// SIMATIC STEP 7 (V5.x) project nef
// CPU: PLC 314C-2 DP
// station: P_ADR_BUS
// station: Hardware
// station: SIMATIC 300(1)
// program: Programma S7(1)

SYMBOL_TABLE
"READ_CLK"	SFC 1	SFC 1	// Read System Clock
"BLKMOV"	SFC 20	SFC 20	// Copy Variables
"FILL"	SFC 21	SFC 21	// Initialize a Memory Area
"CREAT_DB"	SFC 22	SFC 22	// Create Data Block
"DIS_AIRT"	SFC 41	SFC 41	// Delay the Higher Priority Interrupts and Asynchronous Errors
"EN_AIRT"	SFC 42	SFC 42	// Enable Higher Priority Interrupts and Asynchronous Errors
"STP"	SFC 46	SFC 46	// Change the CPU to STOP
"WAIT"	SFC 47	SFC 47	// Delay Execution of the User Program
"RDSYSST"	SFC 51	SFC 51	// Read a System Status List or Partial List
"WR_USMSG"	SFC 52	SFC 52	// Write a User-Defined Diagnostic Event to the Diagnostic Buffer
"TIME_TCK"	SFC 64	SFC 64	// Read the System Time
END_SYMBOL_TABLE

// FB 1: know-how protected block, not included

// FB 2: know-how protected block, not included

// FB 3: know-how protected block, not included

// FB 4: know-how protected block, not included

// FB 5: know-how protected block, not included

// FB 6: know-how protected block, not included

// FB 7: know-how protected block, not included

// FB 9: know-how protected block, not included

// FB 10: know-how protected block, not included

// FB 11: know-how protected block, not included

// FB 15: know-how protected block, not included

// FB 16: know-how protected block, not included

// FB 17: know-how protected block, not included

// FB 18: know-how protected block, not included

// FB 19: know-how protected block, not included

FUNCTION_BLOCK FB 20
VERSION : 2.2
BEGIN
// (block stored without names or comments; labels and parameter names are numbered)
NETWORK
TITLE =
      L     DW#16#87000000;
      LAR1;
      L     80;
      L     W#16#A000;
      +I;
      T     LW 0;
      A      [AR1,P#8.0];
      =     L 0.0;
      L     W [AR1,P#0.0];
      T     LW 2;
      L     W [AR1,P#6.0];
      SLD   16;
      L     B [AR1,P#4.0];
      OD;
      T     LD 4;
      CALL  "WR_USMSG" (
           SEND                     := TRUE,
           EVENTN                   := LW 0,
           INFO1                    := P#L 2.0 INT 1,
           INFO2                    := P#L 4.0 DINT 1,
           RET_VAL                  := LW 8);
END_FUNCTION_BLOCK

FUNCTION_BLOCK FB 100
VERSION : 0.0
BEGIN
// body was compiled from an SCL source; compiled code not shown
END_FUNCTION_BLOCK

FUNCTION_BLOCK FB 101
VERSION : 0.0
BEGIN
// body was compiled from an SCL source; compiled code not shown
END_FUNCTION_BLOCK

// FB 102: know-how protected block, not included

FUNCTION_BLOCK FB 103
VERSION : 0.0
BEGIN
// body was compiled from an SCL source; compiled code not shown
END_FUNCTION_BLOCK

// FB 104: know-how protected block, not included

FUNCTION_BLOCK FB 106
VERSION : 0.0
BEGIN
// body was compiled from an SCL source; compiled code not shown
END_FUNCTION_BLOCK

FUNCTION_BLOCK FB 107
VERSION : 0.0
BEGIN
// body was compiled from an SCL source; compiled code not shown
END_FUNCTION_BLOCK

FUNCTION_BLOCK FB 108
VERSION : 0.0
BEGIN
// body was compiled from an SCL source; compiled code not shown
END_FUNCTION_BLOCK

FUNCTION_BLOCK FB 109
VERSION : 0.0
BEGIN
// body was compiled from an SCL source; compiled code not shown
END_FUNCTION_BLOCK

FUNCTION_BLOCK FB 110
VERSION : 0.0
BEGIN
// body was compiled from an SCL source; compiled code not shown
END_FUNCTION_BLOCK

FUNCTION_BLOCK FB 111
VERSION : 0.0
BEGIN
// body was compiled from an SCL source; compiled code not shown
END_FUNCTION_BLOCK

FUNCTION_BLOCK FB 114
VERSION : 0.0
BEGIN
// body was compiled from an SCL source; compiled code not shown
END_FUNCTION_BLOCK

FUNCTION_BLOCK FB 115
VERSION : 0.0
BEGIN
// body was compiled from an SCL source; compiled code not shown
END_FUNCTION_BLOCK

// FB 116: know-how protected block, not included

FUNCTION_BLOCK FB 117
VERSION : 0.0
BEGIN
// body was compiled from an SCL source; compiled code not shown
END_FUNCTION_BLOCK

FUNCTION_BLOCK FB 118
VERSION : 0.0
BEGIN
// body was compiled from an SCL source; compiled code not shown
END_FUNCTION_BLOCK

FUNCTION_BLOCK FB 119
VERSION : 0.0
BEGIN
// body was compiled from an SCL source; compiled code not shown
END_FUNCTION_BLOCK

FUNCTION_BLOCK FB 120
VERSION : 0.0
BEGIN
// body was compiled from an SCL source; compiled code not shown
END_FUNCTION_BLOCK

// FB 122: know-how protected block, not included

FUNCTION_BLOCK FB 123
VERSION : 0.0
BEGIN
// body was compiled from an SCL source; compiled code not shown
END_FUNCTION_BLOCK

FUNCTION_BLOCK FB 124
VERSION : 0.0
BEGIN
// body was compiled from an SCL source; compiled code not shown
END_FUNCTION_BLOCK

FUNCTION_BLOCK FB 125
VERSION : 0.0
BEGIN
// body was compiled from an SCL source; compiled code not shown
END_FUNCTION_BLOCK

FUNCTION_BLOCK FB 126
VERSION : 0.0
BEGIN
// body was compiled from an SCL source; compiled code not shown
END_FUNCTION_BLOCK

FUNCTION_BLOCK FB 127
VERSION : 0.0
BEGIN
// body was compiled from an SCL source; compiled code not shown
END_FUNCTION_BLOCK

FUNCTION_BLOCK FB 131
VERSION : 0.0
BEGIN
// body was compiled from an SCL source; compiled code not shown
END_FUNCTION_BLOCK

FUNCTION_BLOCK FB 132
VERSION : 0.0
BEGIN
// body was compiled from an SCL source; compiled code not shown
END_FUNCTION_BLOCK

FUNCTION_BLOCK FB 133
VERSION : 0.0
BEGIN
// body was compiled from an SCL source; compiled code not shown
END_FUNCTION_BLOCK

FUNCTION_BLOCK FB 135
VERSION : 0.0
BEGIN
// body was compiled from an SCL source; compiled code not shown
END_FUNCTION_BLOCK

FUNCTION_BLOCK FB 138
VERSION : 0.0
BEGIN
// body was compiled from an SCL source; compiled code not shown
END_FUNCTION_BLOCK

FUNCTION_BLOCK FB 144
VERSION : 0.0
BEGIN
// body was compiled from an SCL source; compiled code not shown
END_FUNCTION_BLOCK

FUNCTION_BLOCK FB 148
VERSION : 0.0
BEGIN
// body was compiled from an SCL source; compiled code not shown
END_FUNCTION_BLOCK

FUNCTION_BLOCK FB 189
AUTHOR : mogs
NAME : s_remind
VERSION : 1.3
BEGIN
// (block stored without names or comments; labels and parameter names are numbered)
NETWORK
TITLE =
      A     DIX 1.0;
      =     L 12.0;
      A     L 12.0;
      A     DIX 172.1;
      R     DIX 172.1;
      R     DIX 173.0;
      A     L 12.0;
      A     DIX 172.0;
      R     DIX 172.0;
      R     DIX 172.7;
      A     L 12.0;
      BLD   102;
      R     DIX 172.2;
NETWORK
TITLE =
      A     DIX 1.1;
      =     L 12.0;
      A     L 12.0;
      A     DIX 172.1;
      R     DIX 172.1;
      S     DIX 173.0;
      A     L 12.0;
      A     DIX 172.0;
      S     DIX 172.7;
      R     DIX 172.0;
      A     L 12.0;
      BLD   102;
      R     DIX 172.3;
NETWORK
TITLE =
      A     DIX 172.0;
      A(;
      L     DIW 2;
      L     0;
      >I;
      );
      =     DIX 18.0;
NETWORK
TITLE =
      A     DIX 172.1;
      A(;
      L     DIW 2;
      L     0;
      >I;
      );
      =     DIX 18.1;
NETWORK
TITLE =
      A     DIX 0.0;
      FP    DIX 172.6;
      =     L 12.0;
      A     L 12.0;
      A     DIX 172.7;
      S     DIX 172.0;
      A     L 12.0;
      A     DIX 173.0;
      S     DIX 172.1;
NETWORK
TITLE =
      BLD   7;
      L     0;
      T     LW 13;
      L     P#V 0.0;
      T     LD 15;
      UC    "READ_CLK";
      {     P#L 8.0, P#L 13.0 };
      BLD   8;
      CLR;
      =     L 10.2;
      =     DIX 173.2;
      =     L 10.1;
      L     LB 5;
      L     DIB 59;
      ==I;
      JC    M001;
      TAK;
      T     DIB 59;
      =     L 10.2;
M001: L     LB 4;
      L     DIB 55;
      ==I;
      JC    M002;
      TAK;
      T     DIB 55;
      =     DIX 173.2;
M002: L     LB 3;
      L     DIB 54;
      ==I;
      JC    M003;
      T     DIB 54;
      =     L 10.1;
M003: L     LB 4;
      BTI;
      T     DIB 65;
      L     LB 3;
      BTI;
      T     DIB 64;
      L     LB 2;
      BTI;
      T     DIB 63;
      L     LB 1;
      BTI;
      T     DIB 62;
      L     LB 0;
      BTI;
      T     DIB 61;
      AN    L 10.2;
      AN    DIX 173.2;
      AN    L 10.1;
      BEC;
NETWORK
TITLE =
// (network holds code this reader does not know; not shown)
NETWORK
TITLE =
// (network holds code this reader does not know; not shown)
NETWORK
TITLE =
// (network holds code this reader does not know; not shown)
NETWORK
TITLE =
M009: NOP   0;
NETWORK
TITLE =
      A     DIX 173.1;
      =     L 12.0;
      A     L 12.0;
      A     DIX 0.3;
      JNB   M010;
      L     0;
      T     DIW 72;
      SET;
      SAVE;
      CLR;
M010: A     BR;
      S     DIX 172.5;
      R     DIX 0.3;
      A     L 12.0;
      A     DIX 172.5;
      A(;
      L     DIW 72;
      L     DIW 4;
      >=I;
      );
      R     DIX 172.5;
NETWORK
TITLE =
      A     DIX 172.5;
      A     DIX 0.0;
      A     DIX 173.2;
      JNB   M011;
      L     DIW 72;
      L     1;
      +I;
      T     DIW 72;
M011: NOP   0;
NETWORK
TITLE =
      BEU;
END_FUNCTION_BLOCK

FUNCTION_BLOCK FB 201
AUTHOR : Duesed
NAME : M_Dek
VERSION : 0.1
BEGIN
// (block stored without names or comments; labels and parameter names are numbered)
NETWORK
TITLE =
      A     DIX [AR2,P#6.0];
      JC    M001;
      JU    M003;
M001: T     LD 27;
      TAK;
      T     LD 31;
      L     DIW [AR2,P#4.0];
      T     LW 35;
      L     LD 31;
      L     LD 27;
      OPN   DB [LW 35];
      L     P#0.0;
      LAR1;
      L     95;
M002: T     LW 4;
      L     0;
      T     DBD [AR1,P#0.0];
      +AR1  P#4.0;
      L     LW 4;
      LOOP  M002;
      CLR;
      =     DIX [AR2,P#8.0];
      =     DIX [AR2,P#8.1];
      =     DIX [AR2,P#8.2];
      L     0;
      T     DID [AR2,P#30.0];
      T     DID [AR2,P#34.0];
      T     DID [AR2,P#38.0];
      T     DID [AR2,P#42.0];
      T     DID [AR2,P#46.0];
      L     -1;
      T     DIW [AR2,P#20.0];
      T     DIW [AR2,P#22.0];
      T     DIW [AR2,P#24.0];
      T     DIW [AR2,P#26.0];
      T     DIW [AR2,P#28.0];
M003: A     DIX [AR2,P#6.1];
      JCN   M032;
      R     DIX [AR2,P#8.4];
      L     -1;
      T     DIW [AR2,P#10.0];
      T     DIW [AR2,P#12.0];
      T     DIW [AR2,P#14.0];
      T     DIW [AR2,P#16.0];
      T     DIW [AR2,P#18.0];
      T     LD 27;
      TAK;
      T     LD 31;
      L     DIW [AR2,P#4.0];
      T     LW 35;
      L     LD 31;
      L     LD 27;
      OPN   DB [LW 35];
      L     0;
      T     LW 24;
M004: L     LW 24;
      JL    M005;
      JU    M006;
      JU    M007;
      JU    M008;
      JU    M009;
      JU    M010;
M005: CLR;
      =     L 26.1;
      JU    M013;
M006: CLR;
      =     L 26.1;
      L     DIW [AR2,P#20.0];
      L     DIW [AR2,P#22.0];
      ==I;
      S     L 26.1;
      L     DIW [AR2,P#20.0];
      L     DIW [AR2,P#24.0];
      ==I;
      S     L 26.1;
      L     DIW [AR2,P#20.0];
      L     DIW [AR2,P#26.0];
      ==I;
      S     L 26.1;
      L     DIW [AR2,P#20.0];
      L     DIW [AR2,P#28.0];
      ==I;
      S     L 26.1;
      L     DIW [AR2,P#20.0];
      T     LD 20;
      L     DID [AR2,P#30.0];
      T     LD 14;
      JU    M011;
M007: CLR;
      =     L 26.1;
      L     DIW [AR2,P#22.0];
      L     DIW [AR2,P#24.0];
      ==I;
      S     L 26.1;
      L     DIW [AR2,P#22.0];
      L     DIW [AR2,P#26.0];
      ==I;
      S     L 26.1;
      L     DIW [AR2,P#22.0];
      L     DIW [AR2,P#28.0];
      ==I;
      S     L 26.1;
      L     DIW [AR2,P#22.0];
      T     LD 20;
      L     DID [AR2,P#34.0];
      T     LD 14;
      JU    M011;
M008: CLR;
      =     L 26.1;
      L     DIW [AR2,P#24.0];
      L     DIW [AR2,P#26.0];
      ==I;
      S     L 26.1;
      L     DIW [AR2,P#24.0];
      L     DIW [AR2,P#28.0];
      ==I;
      S     L 26.1;
      L     DIW [AR2,P#24.0];
      T     LD 20;
      L     DID [AR2,P#38.0];
      T     LD 14;
      JU    M011;
M009: CLR;
      =     L 26.1;
      L     DIW [AR2,P#26.0];
      L     DIW [AR2,P#28.0];
      ==I;
      S     L 26.1;
      L     DIW [AR2,P#26.0];
      T     LD 20;
      L     DID [AR2,P#42.0];
      T     LD 14;
      JU    M011;
M010: CLR;
      =     L 26.1;
      L     DIW [AR2,P#28.0];
      T     LD 20;
      L     DID [AR2,P#46.0];
      T     LD 14;
      JU    M011;
NETWORK
TITLE =
M011: L     LD 20;
      L     -1;
      ==I;
      JC    M012;
      A     L 26.1;
      S     DIX [AR2,P#8.3];
      JC    M012;
      L     LD 20;
      L     999;
      >I;
      JC    M012;
M012: L     LW 24;
      INC   1;
      T     LW 24;
      JU    M004;
M013: NOP   0;
NETWORK
TITLE =
      L     0;
      T     LW 24;
M014: L     LW 24;
      JL    M015;
      JU    M016;
      JU    M017;
      JU    M018;
      JU    M019;
      JU    M020;
M015: BEU;
M016: T     LD 27;
      TAK;
      T     LD 31;
      L     DIW [AR2,P#0.0];
      T     LW 35;
      L     LD 31;
      L     LD 27;
      OPN   DB [LW 35];
      A     DBX 66.0;
      =     L 26.0;
      AN    DBX 58.0;
      JC    M031;
      L     DBW 68;
      T     LW 18;
      L     DBD 70;
      T     LD 20;
      JU    M021;
M017: T     LD 27;
      TAK;
      T     LD 31;
      L     DIW [AR2,P#0.0];
      T     LW 35;
      L     LD 31;
      L     LD 27;
      OPN   DB [LW 35];
      A     DBX 66.1;
      =     L 26.0;
      AN    DBX 58.1;
      JC    M031;
      L     DBW 74;
      T     LW 18;
      L     DBD 76;
      T     LD 20;
      JU    M021;
M018: T     LD 27;
      TAK;
      T     LD 31;
      L     DIW [AR2,P#0.0];
      T     LW 35;
      L     LD 31;
      L     LD 27;
      OPN   DB [LW 35];
      A     DBX 66.2;
      =     L 26.0;
      AN    DBX 58.2;
      JC    M031;
      L     DBW 80;
      T     LW 18;
      L     DBD 82;
      T     LD 20;
      JU    M021;
M019: T     LD 27;
      TAK;
      T     LD 31;
      L     DIW [AR2,P#0.0];
      T     LW 35;
      L     LD 31;
      L     LD 27;
      OPN   DB [LW 35];
      A     DBX 66.3;
      =     L 26.0;
      AN    DBX 58.3;
      JC    M031;
      L     DBW 86;
      T     LW 18;
      L     DBD 88;
      T     LD 20;
      JU    M021;
M020: T     LD 27;
      TAK;
      T     LD 31;
      L     DIW [AR2,P#0.0];
      T     LW 35;
      L     LD 31;
      L     LD 27;
      OPN   DB [LW 35];
      A     DBX 66.4;
      =     L 26.0;
      AN    DBX 58.4;
      JC    M031;
      L     DBW 92;
      T     LW 18;
      L     DBD 94;
      T     LD 20;
      JU    M021;
NETWORK
TITLE =
M021: L     LW 18;
      L     0;
      ==I;
      JC    M024;
      L     LW 18;
      L     DIW [AR2,P#2.0];
      >I;
      JC    M022;
      L     LD 20;
      L     3;
      ==I;
      JC    M023;
      L     LD 20;
      L     4;
      ==I;
      JC    M023;
      L     LD 20;
      L     5;
      ==I;
      JC    M023;
      L     LD 20;
      L     40;
      ==I;
      JC    M023;
      L     LD 20;
      L     41;
      ==I;
      JC    M023;
      L     LD 20;
      L     42;
      ==I;
      JC    M023;
      L     LD 20;
      L     70;
      ==I;
      JC    M031;
M022: S     DIX [AR2,P#8.2];
      JU    M031;
M023: L     LW 18;
      L     100;
      *I;
      L     LD 20;
      +I;
      T     LD 20;
M024: L     LD 20;
      L     999;
      >D;
      S     DIX [AR2,P#8.1];
      JC    M031;
      L     LD 20;
      L     8;
      /I;
      T     LD 6;
      L     LD 6;
      SLD   16;
      SRD   16;
      T     LW 10;
      L     LD 6;
      SRD   16;
      T     LW 12;
      L     LW 10;
      SLW   3;
      L     LW 12;
      OW;
      L     DW#16#4000000;
      OW;
      LAR1;
      T     LD 14;
      T     LD 27;
      TAK;
      T     LD 31;
      L     DIW [AR2,P#4.0];
      T     LW 35;
      L     LD 31;
      L     LD 27;
      OPN   DB [LW 35];
      SET;
      =     DBX [AR1,P#0.0];
      S     DIX [AR2,P#8.4];
      A     L 26.0;
      =     DBX [AR1,P#252.0];
      L     LW 24;
      JL    M025;
      JU    M026;
      JU    M027;
      JU    M028;
      JU    M029;
      JU    M030;
M025: JU    M031;
M026: L     LD 14;
      T     DID [AR2,P#30.0];
      L     LD 20;
      T     DIW [AR2,P#20.0];
      T     DIW [AR2,P#10.0];
      JU    M031;
M027: L     LD 14;
      T     DID [AR2,P#34.0];
      L     LD 20;
      T     DIW [AR2,P#22.0];
      T     DIW [AR2,P#12.0];
      JU    M031;
M028: L     LD 14;
      T     DID [AR2,P#38.0];
      L     LD 20;
      T     DIW [AR2,P#24.0];
      T     DIW [AR2,P#14.0];
      JU    M031;
M029: L     LD 14;
      T     DID [AR2,P#42.0];
      L     LD 20;
      T     DIW [AR2,P#26.0];
      T     DIW [AR2,P#16.0];
      JU    M031;
M030: L     LD 14;
      T     DID [AR2,P#46.0];
      L     LD 20;
      T     DIW [AR2,P#28.0];
      T     DIW [AR2,P#18.0];
      JU    M031;
M031: L     LW 24;
      INC   1;
      T     LW 24;
      JU    M014;
M032: NOP   0;
NETWORK
TITLE =
      AN    DIX [AR2,P#6.1];
      JCN   M038;
      L     DIW [AR2,P#20.0];
      L     -1;
      ==I;
      JC    M033;
      TAK;
      L     999;
      >I;
      JC    M033;
      T     LD 27;
      TAK;
      T     LD 31;
      L     DIW [AR2,P#4.0];
      T     LW 35;
      L     LD 31;
      L     LD 27;
      OPN   DB [LW 35];
      L     DID [AR2,P#30.0];
      LAR1;
      AN    DBX [AR1,P#126.0];
      S     DIX [AR2,P#8.0];
      CLR;
      =     DBX [AR1,P#0.0];
      =     DBX [AR1,P#126.0];
      =     DBX [AR1,P#252.0];
M033: NOP   0;
      L     0;
      T     DID [AR2,P#30.0];
      L     -1;
      T     DIW [AR2,P#20.0];
      L     DIW [AR2,P#22.0];
      L     -1;
      ==I;
      JC    M034;
      TAK;
      L     999;
      >I;
      JC    M034;
      T     LD 27;
      TAK;
      T     LD 31;
      L     DIW [AR2,P#4.0];
      T     LW 35;
      L     LD 31;
      L     LD 27;
      OPN   DB [LW 35];
      L     DID [AR2,P#34.0];
      LAR1;
      AN    DBX [AR1,P#126.0];
      S     DIX [AR2,P#8.0];
      CLR;
      =     DBX [AR1,P#0.0];
      =     DBX [AR1,P#126.0];
      =     DBX [AR1,P#252.0];
M034: NOP   0;
      L     0;
      T     DID [AR2,P#34.0];
      L     -1;
      T     DIW [AR2,P#22.0];
      L     DIW [AR2,P#24.0];
      L     -1;
      ==I;
      JC    M035;
      TAK;
      L     999;
      >I;
      JC    M035;
      T     LD 27;
      TAK;
      T     LD 31;
      L     DIW [AR2,P#4.0];
      T     LW 35;
      L     LD 31;
      L     LD 27;
      OPN   DB [LW 35];
      L     DID [AR2,P#38.0];
      LAR1;
      AN    DBX [AR1,P#126.0];
      S     DIX [AR2,P#8.0];
      CLR;
      =     DBX [AR1,P#0.0];
      =     DBX [AR1,P#126.0];
      =     DBX [AR1,P#252.0];
M035: NOP   0;
      L     0;
      T     DID [AR2,P#38.0];
      L     -1;
      T     DIW [AR2,P#24.0];
      L     DIW [AR2,P#26.0];
      L     -1;
      ==I;
      JC    M036;
      TAK;
      L     999;
      >I;
      JC    M036;
      T     LD 27;
      TAK;
      T     LD 31;
      L     DIW [AR2,P#4.0];
      T     LW 35;
      L     LD 31;
      L     LD 27;
      OPN   DB [LW 35];
      L     DID [AR2,P#42.0];
      LAR1;
      AN    DBX [AR1,P#126.0];
      S     DIX [AR2,P#8.0];
      CLR;
      =     DBX [AR1,P#0.0];
      =     DBX [AR1,P#126.0];
      =     DBX [AR1,P#252.0];
M036: NOP   0;
      L     0;
      T     DID [AR2,P#42.0];
      L     -1;
      T     DIW [AR2,P#26.0];
      L     DIW [AR2,P#28.0];
      L     -1;
      ==I;
      JC    M037;
      TAK;
      L     999;
      >I;
      JC    M037;
      T     LD 27;
      TAK;
      T     LD 31;
      L     DIW [AR2,P#4.0];
      T     LW 35;
      L     LD 31;
      L     LD 27;
      OPN   DB [LW 35];
      L     DID [AR2,P#46.0];
      LAR1;
      AN    DBX [AR1,P#126.0];
      S     DIX [AR2,P#8.0];
      CLR;
      =     DBX [AR1,P#0.0];
      =     DBX [AR1,P#126.0];
      =     DBX [AR1,P#252.0];
M037: NOP   0;
      L     0;
      T     DID [AR2,P#46.0];
      L     -1;
      T     DIW [AR2,P#28.0];
M038: NOP   0;
END_FUNCTION_BLOCK

FUNCTION_BLOCK FB 203
VERSION : 0.0
BEGIN
// body was compiled from an SCL source; compiled code not shown
END_FUNCTION_BLOCK

FUNCTION_BLOCK FB 204
VERSION : 0.0
BEGIN
// body was compiled from an SCL source; compiled code not shown
END_FUNCTION_BLOCK

FUNCTION_BLOCK FB 205
VERSION : 0.0
BEGIN
// body was compiled from an SCL source; compiled code not shown
END_FUNCTION_BLOCK

FUNCTION_BLOCK FB 206
VERSION : 0.0
BEGIN
// body was compiled from an SCL source; compiled code not shown
END_FUNCTION_BLOCK

FUNCTION_BLOCK FB 208
VERSION : 0.0
BEGIN
// body was compiled from an SCL source; compiled code not shown
END_FUNCTION_BLOCK

FUNCTION_BLOCK FB 209
VERSION : 0.0
BEGIN
// body was compiled from an SCL source; compiled code not shown
END_FUNCTION_BLOCK

FUNCTION_BLOCK FB 214
AUTHOR : BI_HSc
VERSION : 0.1
BEGIN
// (block stored without names or comments; labels and parameter names are numbered)
NETWORK
TITLE =
      A     M 0.5;
      JCN   M001;
      OPN   DB 2;
      L     DBLG;
      L     180;
      -I;
      L     8;
      /I;
      OPN   DB 214;
      T     DIW [AR2,P#160.0];
M001: NOP   0;
NETWORK
TITLE =
      OPN   DB 2;
      L     P#180.0;
      LAR1;
      L     P#0.0;
      OPN   DB 214;
      L     P#0.0;
      LAR2;
      SET;
      R     M 2.3;
      R     M 2.4;
      R     M 2.6;
      R     M 2.7;
      R     M 3.0;
      L     DIW [AR2,P#160.0];
M002: T     LW 0;
      OPN   DB 2;
      L     DBD [AR1,P#0.0];
      T     LD 2;
      L     0;
      <>D;
      S     M 2.3;
      TAK;
      OPN   DB 214;
      L     DBD [AR2,P#0.0];
      XOD;
      L     LD 2;
      AD;
      L     0;
      <>D;
      S     M 2.6;
      L     LD 2;
      T     DBD [AR2,P#0.0];
      +AR1  P#4.0;
      +AR2  P#4.0;
      OPN   DB 2;
      L     DBD [AR1,P#0.0];
      T     LD 2;
      L     0;
      <>D;
      S     M 2.4;
      TAK;
      OPN   DB 214;
      L     DBD [AR2,P#0.0];
      XOD;
      L     LD 2;
      AD;
      L     0;
      <>D;
      S     M 2.7;
      L     LD 2;
      T     DBD [AR2,P#0.0];
      +AR1  P#4.0;
      +AR2  P#4.0;
      L     LW 0;
      LOOP  M002;
      A     DB10.DBX 109.0;
      AN    M 2.5;
      S     M 3.0;
      A     DB10.DBX 109.0;
      =     M 2.5;
END_FUNCTION_BLOCK

FUNCTION_BLOCK FB 219
VERSION : 0.0
BEGIN
// body was compiled from an SCL source; compiled code not shown
END_FUNCTION_BLOCK

FUNCTION_BLOCK FB 220
VERSION : 0.0
BEGIN
// body was compiled from an SCL source; compiled code not shown
END_FUNCTION_BLOCK

FUNCTION_BLOCK FB 221
VERSION : 0.0
BEGIN
// body was compiled from an SCL source; compiled code not shown
END_FUNCTION_BLOCK

FUNCTION_BLOCK FB 240
VERSION : 0.0
BEGIN
// body was compiled from an SCL source; compiled code not shown
END_FUNCTION_BLOCK

FUNCTION_BLOCK FB 250
VERSION : 0.0
BEGIN
// body was compiled from an SCL source; compiled code not shown
END_FUNCTION_BLOCK

FUNCTION_BLOCK FB 252
VERSION : 0.0
BEGIN
// body was compiled from an SCL source; compiled code not shown
END_FUNCTION_BLOCK

FUNCTION_BLOCK FB 253
VERSION : 0.0
BEGIN
// body was compiled from an SCL source; compiled code not shown
END_FUNCTION_BLOCK

// FC 1: know-how protected block, not included

// FC 2: know-how protected block, not included

// FC 3: know-how protected block, not included

// FC 4: know-how protected block, not included

// FC 6: know-how protected block, not included

// FC 7: know-how protected block, not included

// FC 8: know-how protected block, not included

// FC 9: know-how protected block, not included

// FC 10: know-how protected block, not included

// FC 11: know-how protected block, not included

FUNCTION FC 12 : VOID
AUTHOR : NUMERIK
FAMILY : _800D
NAME : Basics
VERSION : 4.0
BEGIN
// (block stored without names or comments; labels and parameter names are numbered)
END_FUNCTION

// FC 13: know-how protected block, not included

// FC 14: know-how protected block, not included

// FC 15: know-how protected block, not included

// FC 16: know-how protected block, not included

// FC 17: know-how protected block, not included

// FC 18: know-how protected block, not included

FUNCTION FC 19 : VOID
AUTHOR : NUMERIK
FAMILY : _800D
NAME : MCP_IFM
VERSION : 6.1
BEGIN
// (block stored without names or comments; labels and parameter names are numbered)
NETWORK
TITLE =
// (network holds code this reader does not know; not shown)
END_FUNCTION

// FC 20: know-how protected block, not included

// FC 21: know-how protected block, not included

// FC 22: know-how protected block, not included

FUNCTION FC 24 : VOID
AUTHOR : NUMERIK
FAMILY : _800D
NAME : MCP_IFM2
VERSION : 6.1
BEGIN
// (block stored without names or comments; labels and parameter names are numbered)
NETWORK
TITLE =
// (network holds code this reader does not know; not shown)
END_FUNCTION

FUNCTION FC 25 : VOID
AUTHOR : NUMERIK
FAMILY : _800D
NAME : MCP_IFT
VERSION : 6.1
BEGIN
// (block stored without names or comments; labels and parameter names are numbered)
NETWORK
TITLE =
// (network holds code this reader does not know; not shown)
END_FUNCTION

FUNCTION FC 26 : VOID
AUTHOR : NUMERIK
FAMILY : _800D
NAME : HPU_MCP
VERSION : 6.2
BEGIN
// (block stored without names or comments; labels and parameter names are numbered)
NETWORK
TITLE =
// (network holds code this reader does not know; not shown)
END_FUNCTION

FUNCTION FC 30 : VOID
VERSION : 0.0
BEGIN
// body was compiled from another editor; compiled code not shown
END_FUNCTION

FUNCTION FC 31 : VOID
VERSION : 0.0
BEGIN
// body was compiled from another editor; compiled code not shown
END_FUNCTION

FUNCTION FC 32 : VOID
VERSION : 0.0
BEGIN
// body was compiled from another editor; compiled code not shown
END_FUNCTION

FUNCTION FC 33 : VOID
VERSION : 0.0
BEGIN
// body was compiled from another editor; compiled code not shown
END_FUNCTION

// FC 34: know-how protected block, not included

// FC 35: know-how protected block, not included

FUNCTION FC 119 : VOID
VERSION : 0.0
BEGIN
// body was compiled from an SCL source; compiled code not shown
END_FUNCTION

FUNCTION FC 123 : VOID
NAME : TEST2
VERSION : 0.0
BEGIN
// (block stored without names or comments; labels and parameter names are numbered)
NETWORK
TITLE =
      CLR;
      =     #PARAM7;
      L     0;
      T     #PARAM8;
      AN    #PARAM1;
      BEC;
      SET;
      S     L 0.0;
      L     -1;
      T     #PARAM6;
NETWORK
TITLE =
      L     #PARAM3;
      T     LW 2;
      OPN   DB [LW 2];
      L     DBLG;
      L     2;
      -D;
      T     LW 4;
      L     #PARAM4;
      L     LW 4;
      >D;
      L     2;
      JC    M002;
      A     #PARAM2;
      JC    M001;
NETWORK
TITLE =
      L     #PARAM4;
      SLW   3;
      LAR1;
      L     DBW [AR1,P#0.0];
      T     LW 6;
      T     #PARAM6;
      CALL  FC 21 (
           $1                       := P#L 0.0,
           $2                       := B#16#4,
           $3                       := P#L 6.0 WORD 1,
           $4                       := 1020,
           $5                       := -1,
           $6                       := #PARAM7,
           $7                       := #PARAM8);
      L     #PARAM8;
      A     #PARAM7;
      JC    M002;
      JU    M003;
NETWORK
TITLE =
M001: L     #PARAM4;
      SLW   3;
      LAR1;
      L     #PARAM5;
      T     DBW [AR1,P#0.0];
      JU    M003;
NETWORK
TITLE =
M002: SET;
      =     #PARAM7;
      T     #PARAM8;
M003: NOP   0;
END_FUNCTION

FUNCTION FC 200 : VOID
VERSION : 0.0
BEGIN
// body was compiled from an SCL source; compiled code not shown
END_FUNCTION

FUNCTION FC 201 : VOID
VERSION : 0.0
BEGIN
// body was compiled from an SCL source; compiled code not shown
END_FUNCTION

// FC 202: know-how protected block, not included

// FC 225: know-how protected block, not included

// FC 226: know-how protected block, not included

FUNCTION FC 241 : VOID
AUTHOR : RuestGeh
FAMILY : SPL
VERSION : 3.0
BEGIN
// (block stored without names or comments; labels and parameter names are numbered)
NETWORK
TITLE =
      L     P##PARAM4;
      LAR1;
      L     P##PARAM13;
      LAR2;
      L     DB5.DBW 24;
      L     #PARAM3;
      <I;
      JC    M054;
      L     0;
      >I;
      JCN   M054;
      TAK;
      L     8;
      >I;
      JC    M054;
      A     #PARAM14;
      R     #PARAM14;
      A     #PARAM2;
      FP     [AR2,P#1.6];
      JC    M055;
      A     #PARAM1;
      FP     [AR2,P#1.7];
      S      [AR2,P#0.0];
      L     P##PARAM4;
      LAR1;
      L     #PARAM3;
      A      [AR2,P#0.0];
      JC    M001;
      A      [AR2,P#0.1];
      JC    M011;
      A      [AR2,P#0.2];
      JC    M012;
      A      [AR2,P#0.3];
      JC    M022;
      A      [AR2,P#0.4];
      JC    M023;
      A      [AR2,P#0.5];
      JC    M033;
      A      [AR2,P#0.6];
      JC    M043;
      BEU;
NETWORK
TITLE =
M001: L     W [AR1,P#0.0];
      INC   30;
      T     LW 0;
      TAK;
      OPN   DB [LW 0];
      AN    DBX 108.2;
      =      [AR2,P#2.0];
      JCN   M053;
      +AR1  P#2.0;
      +AR2  P#0.1;
      LOOP  M001;
      L     P##PARAM13;
      LAR2;
      L     #PARAM3;
      DEC   1;
      JL    M002;
      JU    M010;
      JU    M009;
      JU    M008;
      JU    M007;
      JU    M006;
      JU    M005;
      JU    M004;
      JU    M003;
M002: JU    M057;
M003: A      [AR2,P#2.7];
M004: A      [AR2,P#2.6];
M005: A      [AR2,P#2.5];
M006: A      [AR2,P#2.4];
M007: A      [AR2,P#2.3];
M008: A      [AR2,P#2.2];
M009: A      [AR2,P#2.1];
M010: A      [AR2,P#2.0];
      A      [AR2,P#0.0];
      R      [AR2,P#0.0];
      S      [AR2,P#0.1];
      BEU;
NETWORK
TITLE =
M011: L     W [AR1,P#0.0];
      INC   30;
      T     LW 0;
      TAK;
      OPN   DB [LW 0];
      A      [AR2,P#0.1];
      S     DBX 23.7;
      +AR1  P#2.0;
      LOOP  M011;
      A      [AR2,P#0.1];
      R      [AR2,P#0.1];
      S      [AR2,P#0.2];
      BEU;
NETWORK
TITLE =
M012: L     W [AR1,P#0.0];
      INC   30;
      T     LW 0;
      TAK;
      OPN   DB [LW 0];
      A     DBX 108.2;
      =      [AR2,P#2.0];
      +AR1  P#2.0;
      +AR2  P#0.1;
      LOOP  M012;
      L     P##PARAM13;
      LAR2;
      L     #PARAM3;
      DEC   1;
      JL    M013;
      JU    M021;
      JU    M020;
      JU    M019;
      JU    M018;
      JU    M017;
      JU    M016;
      JU    M015;
      JU    M014;
M013: JU    M057;
M014: A      [AR2,P#2.7];
M015: A      [AR2,P#2.6];
M016: A      [AR2,P#2.5];
M017: A      [AR2,P#2.4];
M018: A      [AR2,P#2.3];
M019: A      [AR2,P#2.2];
M020: A      [AR2,P#2.1];
M021: A      [AR2,P#2.0];
      A      [AR2,P#0.2];
      R      [AR2,P#0.2];
      S      [AR2,P#0.3];
      BEU;
NETWORK
TITLE =
M022: L     W [AR1,P#0.0];
      INC   30;
      T     LW 0;
      TAK;
      OPN   DB [LW 0];
      A      [AR2,P#0.3];
      R     DBX 23.7;
      +AR1  P#2.0;
      LOOP  M022;
      A      [AR2,P#0.3];
      R      [AR2,P#0.3];
      S      [AR2,P#0.4];
      BEU;
NETWORK
TITLE =
M023: L     W [AR1,P#0.0];
      INC   30;
      T     LW 0;
      TAK;
      OPN   DB [LW 0];
      AN    DBX 108.2;
      =      [AR2,P#2.0];
      +AR1  P#2.0;
      +AR2  P#0.1;
      LOOP  M023;
      L     P##PARAM13;
      LAR2;
      L     #PARAM3;
      DEC   1;
      JL    M024;
      JU    M032;
      JU    M031;
      JU    M030;
      JU    M029;
      JU    M028;
      JU    M027;
      JU    M026;
      JU    M025;
M024: JU    M057;
M025: A      [AR2,P#2.7];
M026: A      [AR2,P#2.6];
M027: A      [AR2,P#2.5];
M028: A      [AR2,P#2.4];
M029: A      [AR2,P#2.3];
M030: A      [AR2,P#2.2];
M031: A      [AR2,P#2.1];
M032: A      [AR2,P#2.0];
      A      [AR2,P#0.4];
      R      [AR2,P#0.4];
      S      [AR2,P#0.5];
      S     #PARAM12;
      BEU;
NETWORK
TITLE =
M033: L     W [AR1,P#0.0];
      INC   30;
      T     LW 0;
      TAK;
      OPN   DB [LW 0];
      A     DBX 108.2;
      =      [AR2,P#3.0];
      +AR1  P#2.0;
      +AR2  P#0.1;
      LOOP  M033;
      L     P##PARAM13;
      LAR2;
      L     #PARAM3;
      DEC   1;
      JL    M034;
      JU    M042;
      JU    M041;
      JU    M040;
      JU    M039;
      JU    M038;
      JU    M037;
      JU    M036;
      JU    M035;
M034: JU    M057;
M035: A      [AR2,P#3.7];
M036: A      [AR2,P#3.6];
M037: A      [AR2,P#3.5];
M038: A      [AR2,P#3.4];
M039: A      [AR2,P#3.3];
M040: A      [AR2,P#3.2];
M041: A      [AR2,P#3.1];
M042: A      [AR2,P#3.0];
      A      [AR2,P#0.5];
      R      [AR2,P#0.5];
      S      [AR2,P#0.6];
      R     #PARAM12;
      BEU;
NETWORK
TITLE =
M043: L     W [AR1,P#0.0];
      INC   30;
      T     LW 0;
      TAK;
      OPN   DB [LW 0];
      AN    DBX 108.2;
      =      [AR2,P#3.0];
      +AR1  P#2.0;
      +AR2  P#0.1;
      LOOP  M043;
      L     P##PARAM13;
      LAR2;
      L     #PARAM3;
      DEC   1;
      JL    M044;
      JU    M052;
      JU    M051;
      JU    M050;
      JU    M049;
      JU    M048;
      JU    M047;
      JU    M046;
      JU    M045;
M044: JU    M057;
M045: A      [AR2,P#3.7];
M046: A      [AR2,P#3.6];
M047: A      [AR2,P#3.5];
M048: A      [AR2,P#3.4];
M049: A      [AR2,P#3.3];
M050: A      [AR2,P#3.2];
M051: A      [AR2,P#3.1];
M052: A      [AR2,P#3.0];
      A      [AR2,P#0.6];
      R      [AR2,P#0.6];
      S     #PARAM14;
      JC    M056;
      BEU;
NETWORK
TITLE =
M053: =     #PARAM15;
      JU    M056;
M054: =     #PARAM16;
      JU    M056;
M055: SET;
      R     #PARAM15;
      R     #PARAM16;
M056: L     #PARAM13;
      L     DW#16#C00000;
      AD;
      T     #PARAM13;
      SET;
      R     #PARAM12;
M057: BE;
END_FUNCTION

FUNCTION FC 243 : VOID
AUTHOR : Gehringe
FAMILY : SPL
VERSION : 3.0
BEGIN
// (block stored without names or comments; labels and parameter names are numbered)
NETWORK
TITLE =
      L     P##PARAM4;
      LAR1;
      L     P##PARAM13;
      LAR2;
      L     DB5.DBW 24;
      L     #PARAM3;
      <I;
      JC    M032;
      L     0;
      >I;
      JCN   M032;
      TAK;
      L     8;
      >I;
      JC    M032;
      A     #PARAM14;
      R     #PARAM14;
      A     #PARAM2;
      FP     [AR2,P#1.6];
      JC    M033;
      A     #PARAM1;
      FP     [AR2,P#1.7];
      S      [AR2,P#0.0];
      L     P##PARAM4;
      LAR1;
      L     #PARAM3;
      A      [AR2,P#0.0];
      JC    M001;
      A      [AR2,P#0.1];
      JC    M011;
      A      [AR2,P#0.2];
      JC    M021;
      BEU;
NETWORK
TITLE =
M001: L     W [AR1,P#0.0];
      INC   30;
      T     LW 0;
      TAK;
      OPN   DB [LW 0];
      AN    DBX 108.2;
      =      [AR2,P#2.0];
      JCN   M031;
      +AR1  P#2.0;
      +AR2  P#0.1;
      LOOP  M001;
      L     P##PARAM13;
      LAR2;
      L     #PARAM3;
      DEC   1;
      JL    M002;
      JU    M010;
      JU    M009;
      JU    M008;
      JU    M007;
      JU    M006;
      JU    M005;
      JU    M004;
      JU    M003;
M002: JU    M035;
M003: A      [AR2,P#2.7];
M004: A      [AR2,P#2.6];
M005: A      [AR2,P#2.5];
M006: A      [AR2,P#2.4];
M007: A      [AR2,P#2.3];
M008: A      [AR2,P#2.2];
M009: A      [AR2,P#2.1];
M010: A      [AR2,P#2.0];
      A      [AR2,P#0.0];
      R      [AR2,P#0.0];
      S      [AR2,P#0.1];
      S     #PARAM12;
      BEU;
NETWORK
TITLE =
M011: L     W [AR1,P#0.0];
      INC   30;
      T     LW 0;
      TAK;
      OPN   DB [LW 0];
      A     DBX 108.2;
      =      [AR2,P#3.0];
      +AR1  P#2.0;
      +AR2  P#0.1;
      LOOP  M011;
      L     P##PARAM13;
      LAR2;
      L     #PARAM3;
      DEC   1;
      JL    M012;
      JU    M020;
      JU    M019;
      JU    M018;
      JU    M017;
      JU    M016;
      JU    M015;
      JU    M014;
      JU    M013;
M012: JU    M035;
M013: A      [AR2,P#3.7];
M014: A      [AR2,P#3.6];
M015: A      [AR2,P#3.5];
M016: A      [AR2,P#3.4];
M017: A      [AR2,P#3.3];
M018: A      [AR2,P#3.2];
M019: A      [AR2,P#3.1];
M020: A      [AR2,P#3.0];
      A      [AR2,P#0.1];
      R      [AR2,P#0.1];
      S      [AR2,P#0.2];
      R     #PARAM12;
      BEU;
NETWORK
TITLE =
M021: L     W [AR1,P#0.0];
      INC   30;
      T     LW 0;
      TAK;
      OPN   DB [LW 0];
      AN    DBX 108.2;
      =      [AR2,P#2.0];
      +AR1  P#2.0;
      +AR2  P#0.1;
      LOOP  M021;
      L     P##PARAM13;
      LAR2;
      L     #PARAM3;
      DEC   1;
      JL    M022;
      JU    M030;
      JU    M029;
      JU    M028;
      JU    M027;
      JU    M026;
      JU    M025;
      JU    M024;
      JU    M023;
M022: JU    M035;
M023: A      [AR2,P#2.7];
M024: A      [AR2,P#2.6];
M025: A      [AR2,P#2.5];
M026: A      [AR2,P#2.4];
M027: A      [AR2,P#2.3];
M028: A      [AR2,P#2.2];
M029: A      [AR2,P#2.1];
M030: A      [AR2,P#2.0];
      A      [AR2,P#0.2];
      R      [AR2,P#0.2];
      S     #PARAM14;
      JC    M034;
      BEU;
NETWORK
TITLE =
M031: =     #PARAM15;
      JU    M034;
M032: =     #PARAM16;
      JU    M034;
M033: SET;
      R     #PARAM15;
      R     #PARAM16;
M034: L     #PARAM13;
      L     DW#16#C00000;
      AD;
      T     #PARAM13;
      SET;
      R     #PARAM12;
M035: BE;
END_FUNCTION

FUNCTION FC 254 : VOID
VERSION : 0.0
BEGIN
// body was compiled from an SCL source; compiled code not shown
END_FUNCTION

// FC 255: know-how protected block, not included

DATA_BLOCK DB 1
VERSION : 0.1
BEGIN
// 14860 bytes; values not shown
END_DATA_BLOCK

DATA_BLOCK DB 2
VERSION : 0.0
UDT 2
BEGIN
END_DATA_BLOCK

DATA_BLOCK DB 3
VERSION : 0.0
BEGIN
// 340 bytes; values not shown
END_DATA_BLOCK

DATA_BLOCK DB 4
AUTHOR : NUMERIK
FAMILY : _800D
NAME : Basics
VERSION : 2.1
BEGIN
// 226 bytes; values not shown
END_DATA_BLOCK

DATA_BLOCK DB 5
AUTHOR : NUMERIK
FAMILY : _800D
NAME : Basics
VERSION : 2.7
BEGIN
// 266 bytes; values not shown
END_DATA_BLOCK

DATA_BLOCK DB 6
VERSION : 0.0
BEGIN
// 272 bytes; values not shown
END_DATA_BLOCK

DATA_BLOCK DB 7
AUTHOR : NUMERIK
FAMILY : _800D
NAME : Basics
VERSION : 2.5
FB 1
BEGIN
END_DATA_BLOCK

DATA_BLOCK DB 8
AUTHOR : NUMERIK
FAMILY : _800D
NAME : Basics
VERSION : 4.3
BEGIN
// 166 bytes; values not shown
END_DATA_BLOCK

DATA_BLOCK DB 10
AUTHOR : NUMERIK
FAMILY : _800D
NAME : Basics
VERSION : 1.1
UDT 10
BEGIN
END_DATA_BLOCK

DATA_BLOCK DB 11
VERSION : 0.0
BEGIN
// 20 bytes; values not shown
END_DATA_BLOCK

DATA_BLOCK DB 15
AUTHOR : NUMERIK
FAMILY : _800D
NAME : Bas_Com
VERSION : 2.1
FB 6
BEGIN
END_DATA_BLOCK

// DB 16: know-how protected block, not included

DATA_BLOCK DB 17
AUTHOR : NUMERIK
FAMILY : _800D
NAME : Basics
VERSION : 2.0
BEGIN
// 4 bytes; values not shown
END_DATA_BLOCK

DATA_BLOCK DB 18
AUTHOR : NUMERIK
FAMILY : _800D
NAME : Basics
VERSION : 6.5
BEGIN
// 190 bytes; values not shown
END_DATA_BLOCK

DATA_BLOCK DB 19
AUTHOR : NUMERIK
FAMILY : _800D
NAME : Basics
VERSION : 2.1
UDT 19
BEGIN
END_DATA_BLOCK

DATA_BLOCK DB 20
VERSION : 0.0
BEGIN
// 896 bytes; values not shown
END_DATA_BLOCK

DATA_BLOCK DB 21
VERSION : 0.0
BEGIN
// 376 bytes; values not shown
END_DATA_BLOCK

DATA_BLOCK DB 31
VERSION : 0.0
UDT 31
BEGIN
END_DATA_BLOCK

DATA_BLOCK DB 32
VERSION : 0.0
UDT 31
BEGIN
END_DATA_BLOCK

DATA_BLOCK DB 33
VERSION : 0.0
UDT 31
BEGIN
END_DATA_BLOCK

DATA_BLOCK DB 34
VERSION : 0.0
UDT 31
BEGIN
END_DATA_BLOCK

DATA_BLOCK DB 35
VERSION : 0.0
UDT 31
BEGIN
END_DATA_BLOCK

DATA_BLOCK DB 40
VERSION : 0.0
UDT 31
BEGIN
END_DATA_BLOCK

DATA_BLOCK DB 71
VERSION : 0.0
BEGIN
// 64 bytes; values not shown
END_DATA_BLOCK

DATA_BLOCK DB 72
VERSION : 0.0
BEGIN
// 52 bytes; values not shown
END_DATA_BLOCK

DATA_BLOCK DB 73
VERSION : 0.0
BEGIN
// 48 bytes; values not shown
END_DATA_BLOCK

DATA_BLOCK DB 74
VERSION : 0.0
BEGIN
// 160 bytes; values not shown
END_DATA_BLOCK

// DB 81: know-how protected block, not included

DATA_BLOCK DB 82
AUTHOR : NUMERIK
NAME : CMM_PLC
VERSION : 0.0
BEGIN
// 182 bytes; values not shown
END_DATA_BLOCK

// DB 83: know-how protected block, not included

DATA_BLOCK DB 84
VERSION : 0.0
BEGIN
// 374 bytes; values not shown
END_DATA_BLOCK

DATA_BLOCK DB 85
VERSION : 0.0
BEGIN
// 280 bytes; values not shown
END_DATA_BLOCK

DATA_BLOCK DB 86
VERSION : 0.0
BEGIN
// 278 bytes; values not shown
END_DATA_BLOCK

DATA_BLOCK DB 87
VERSION : 0.0
BEGIN
// 316 bytes; values not shown
END_DATA_BLOCK

DATA_BLOCK DB 90
VERSION : 0.0
BEGIN
// 2652 bytes; values not shown
END_DATA_BLOCK

DATA_BLOCK DB 92
VERSION : 0.0
BEGIN
// 198 bytes; values not shown
END_DATA_BLOCK

DATA_BLOCK DB 93
VERSION : 0.0
BEGIN
// 208 bytes; values not shown
END_DATA_BLOCK

DATA_BLOCK DB 97
VERSION : 0.1
BEGIN
// 2410 bytes; values not shown
END_DATA_BLOCK

DATA_BLOCK DB 101
VERSION : 0.0
FB 101
BEGIN
END_DATA_BLOCK

DATA_BLOCK DB 102
AUTHOR : BI_HSc
VERSION : 0.0
FB 102
BEGIN
END_DATA_BLOCK

DATA_BLOCK DB 103
VERSION : 0.0
FB 103
BEGIN
END_DATA_BLOCK

DATA_BLOCK DB 104
AUTHOR : BI_HSc
VERSION : 0.0
FB 104
BEGIN
END_DATA_BLOCK

DATA_BLOCK DB 106
VERSION : 0.0
FB 106
BEGIN
END_DATA_BLOCK

DATA_BLOCK DB 107
VERSION : 0.0
FB 107
BEGIN
END_DATA_BLOCK

DATA_BLOCK DB 108
VERSION : 0.0
FB 108
BEGIN
END_DATA_BLOCK

DATA_BLOCK DB 109
VERSION : 0.0
FB 109
BEGIN
END_DATA_BLOCK

DATA_BLOCK DB 110
VERSION : 0.0
FB 110
BEGIN
END_DATA_BLOCK

DATA_BLOCK DB 111
VERSION : 0.0
FB 111
BEGIN
END_DATA_BLOCK

DATA_BLOCK DB 114
VERSION : 0.0
FB 114
BEGIN
END_DATA_BLOCK

DATA_BLOCK DB 115
VERSION : 0.0
FB 115
BEGIN
END_DATA_BLOCK

DATA_BLOCK DB 116
AUTHOR : BI_HSc
VERSION : 0.0
FB 116
BEGIN
END_DATA_BLOCK

DATA_BLOCK DB 117
VERSION : 0.0
FB 117
BEGIN
END_DATA_BLOCK

DATA_BLOCK DB 118
VERSION : 0.0
FB 118
BEGIN
END_DATA_BLOCK

DATA_BLOCK DB 119
VERSION : 0.0
FB 119
BEGIN
END_DATA_BLOCK

DATA_BLOCK DB 120
VERSION : 0.0
FB 120
BEGIN
END_DATA_BLOCK

DATA_BLOCK DB 122
AUTHOR : BI_UWe
VERSION : 0.0
FB 122
BEGIN
END_DATA_BLOCK

DATA_BLOCK DB 123
VERSION : 0.0
FB 123
BEGIN
END_DATA_BLOCK

DATA_BLOCK DB 124
VERSION : 0.0
FB 124
BEGIN
END_DATA_BLOCK

DATA_BLOCK DB 125
VERSION : 0.0
FB 125
BEGIN
END_DATA_BLOCK

DATA_BLOCK DB 126
VERSION : 0.0
FB 126
BEGIN
END_DATA_BLOCK

DATA_BLOCK DB 127
VERSION : 0.0
FB 127
BEGIN
END_DATA_BLOCK

DATA_BLOCK DB 131
VERSION : 0.0
FB 131
BEGIN
END_DATA_BLOCK

DATA_BLOCK DB 132
VERSION : 0.0
FB 132
BEGIN
END_DATA_BLOCK

DATA_BLOCK DB 133
VERSION : 0.0
FB 133
BEGIN
END_DATA_BLOCK

DATA_BLOCK DB 135
VERSION : 0.0
FB 135
BEGIN
END_DATA_BLOCK

DATA_BLOCK DB 138
VERSION : 0.0
FB 138
BEGIN
END_DATA_BLOCK

DATA_BLOCK DB 144
VERSION : 0.0
FB 144
BEGIN
END_DATA_BLOCK

DATA_BLOCK DB 148
VERSION : 0.0
FB 148
BEGIN
END_DATA_BLOCK

DATA_BLOCK DB 164
VERSION : 0.0
FB 164
BEGIN
END_DATA_BLOCK

DATA_BLOCK DB 200
VERSION : 0.0
BEGIN
// 32 bytes; values not shown
END_DATA_BLOCK

DATA_BLOCK DB 201
VERSION : 0.0
UDT 201
BEGIN
END_DATA_BLOCK

DATA_BLOCK DB 210
VERSION : 0.0
BEGIN
// 90 bytes; values not shown
END_DATA_BLOCK

DATA_BLOCK DB 214
AUTHOR : BI_HSc
VERSION : 0.1
FB 214
BEGIN
END_DATA_BLOCK

DATA_BLOCK DB 220
VERSION : 0.1
BEGIN
// 2 bytes; values not shown
END_DATA_BLOCK

DATA_BLOCK DB 221
VERSION : 0.0
FB 221
BEGIN
END_DATA_BLOCK

DATA_BLOCK DB 240
VERSION : 0.0
FB 240
BEGIN
END_DATA_BLOCK

DATA_BLOCK DB 250
VERSION : 0.0
FB 250
BEGIN
END_DATA_BLOCK

DATA_BLOCK DB 252
VERSION : 0.0
FB 252
BEGIN
END_DATA_BLOCK

DATA_BLOCK DB 289
AUTHOR : mogs
VERSION : 0.1
FB 189
BEGIN
END_DATA_BLOCK

DATA_BLOCK DB 299
VERSION : 0.0
BEGIN
// 20 bytes; values not shown
END_DATA_BLOCK

DATA_BLOCK DB 300
VERSION : 0.0
FB 100
BEGIN
END_DATA_BLOCK

DATA_BLOCK DB 319
VERSION : 0.0
BEGIN
// 1604 bytes; values not shown
END_DATA_BLOCK

ORGANIZATION_BLOCK OB 1
AUTHOR : BI_HSc
VERSION : 0.1
VAR_TEMP
  TEMP0 : BYTE ;
  TEMP1 : BYTE ;
  TEMP2 : BYTE ;
  TEMP3 : BYTE ;
  TEMP4 : BYTE ;
  TEMP5 : BYTE ;
  TEMP6 : INT ;
  TEMP7 : INT ;
  TEMP8 : INT ;
  TEMP9 : DATE_AND_TIME ;
  TEMP10 : INT ;
END_VAR
BEGIN
NETWORK
TITLE =
      CALL  FC 2;
      L     #TEMP1;
      L     1;
      ==I;
      =     M 0.5;
      L     #TEMP6;
      T     MW 10;
NETWORK
TITLE =
      CALL  FB 214 , DB 214;
      CALL  FC 200;
NETWORK
TITLE =
      CALL  FB 221 , DB 221;
      CALL  FC 30 (
           $1                       := M 0.5);
NETWORK
TITLE =
      CALL  FB 106 , DB 106 (
           DIX 0.0                  := FALSE);
      CALL  FB 101 , DB 101;
      CALL  FC 10 (
           $1                       := FALSE,
           $2                       := DB21.DBX 7.7);
      CALL  FB 240 , DB 240;
END_ORGANIZATION_BLOCK

ORGANIZATION_BLOCK OB 35
VERSION : 0.1
BEGIN
// (block stored without names or comments; labels and parameter names are numbered)
NETWORK
TITLE =
END_ORGANIZATION_BLOCK

ORGANIZATION_BLOCK OB 40
VERSION : 3.2
BEGIN
// (block stored without names or comments; labels and parameter names are numbered)
NETWORK
TITLE =
      CALL  FC 3;
END_ORGANIZATION_BLOCK

ORGANIZATION_BLOCK OB 80
VERSION : 0.0
BEGIN
// (block stored without names or comments; labels and parameter names are numbered)
NETWORK
TITLE =
      L     LD 0;
      T     DB93.DBD 0;
      T     DB93.DBD 56;
      L     LD 4;
      T     DB93.DBD 4;
      T     DB93.DBD 60;
      L     LD 8;
      T     DB93.DBD 8;
      T     DB93.DBD 64;
      L     LD 12;
      T     DB93.DBD 12;
      T     DB93.DBD 68;
      L     LD 16;
      T     DB93.DBD 16;
      T     DB93.DBD 72;
      L     80;
      T     DB93.DBD 50;
      SET;
      S     DB93.DBX 54.0;
      AN    M 0.7;
      BEC;
      CALL  "STP";
END_ORGANIZATION_BLOCK

ORGANIZATION_BLOCK OB 81
VERSION : 0.0
BEGIN
// (block stored without names or comments; labels and parameter names are numbered)
NETWORK
TITLE =
      L     LD 0;
      T     DB93.DBD 0;
      T     DB93.DBD 78;
      L     LD 4;
      T     DB93.DBD 4;
      T     DB93.DBD 82;
      L     LD 8;
      T     DB93.DBD 8;
      T     DB93.DBD 86;
      L     LD 12;
      T     DB93.DBD 12;
      T     DB93.DBD 90;
      L     LD 16;
      T     DB93.DBD 16;
      T     DB93.DBD 94;
      L     81;
      T     DB93.DBD 50;
      L     LB 0;
      L     B#16#39;
      ==I;
      S     DB93.DBX 76.0;
      L     LB 0;
      L     B#16#38;
      ==I;
      R     DB93.DBX 76.0;
      AN    M 0.7;
      BEC;
      CALL  "STP";
END_ORGANIZATION_BLOCK

ORGANIZATION_BLOCK OB 82
VERSION : 0.0
BEGIN
// (block stored without names or comments; labels and parameter names are numbered)
NETWORK
TITLE =
      L     LD 0;
      T     DB93.DBD 0;
      T     DB93.DBD 100;
      L     LD 4;
      T     DB93.DBD 4;
      T     DB93.DBD 104;
      L     LD 8;
      T     DB93.DBD 8;
      T     DB93.DBD 108;
      L     LD 12;
      T     DB93.DBD 12;
      T     DB93.DBD 112;
      L     LD 16;
      T     DB93.DBD 16;
      T     DB93.DBD 116;
      L     82;
      T     DB93.DBD 50;
      L     LB 0;
      L     B#16#39;
      ==I;
      S     DB93.DBX 98.0;
      L     LB 0;
      L     B#16#38;
      ==I;
      R     DB93.DBX 98.0;
      AN    M 0.7;
      BEC;
      CALL  "STP";
END_ORGANIZATION_BLOCK

ORGANIZATION_BLOCK OB 85
VERSION : 0.0
BEGIN
// (block stored without names or comments; labels and parameter names are numbered)
NETWORK
TITLE =
      L     LD 0;
      T     DB93.DBD 0;
      T     DB93.DBD 122;
      L     LD 4;
      T     DB93.DBD 4;
      T     DB93.DBD 126;
      L     LD 8;
      T     DB93.DBD 8;
      T     DB93.DBD 130;
      L     LD 12;
      T     DB93.DBD 12;
      T     DB93.DBD 134;
      L     LD 16;
      T     DB93.DBD 16;
      T     DB93.DBD 138;
      L     85;
      T     DB93.DBD 50;
      SET;
      S     DB93.DBX 120.0;
      AN    M 0.7;
      BEC;
      CALL  "STP";
END_ORGANIZATION_BLOCK

ORGANIZATION_BLOCK OB 86
VERSION : 0.0
BEGIN
// (block stored without names or comments; labels and parameter names are numbered)
NETWORK
TITLE =
      L     LD 0;
      T     DB93.DBD 0;
      T     DB93.DBD 144;
      L     LD 4;
      T     DB93.DBD 4;
      T     DB93.DBD 148;
      L     LD 8;
      T     DB93.DBD 8;
      T     DB93.DBD 152;
      L     LD 12;
      T     DB93.DBD 12;
      T     DB93.DBD 156;
      L     LD 16;
      T     DB93.DBD 16;
      T     DB93.DBD 160;
      L     86;
      T     DB93.DBD 50;
      L     LB 0;
      L     B#16#39;
      ==I;
      S     DB93.DBX 142.0;
      L     LB 0;
      L     B#16#38;
      ==I;
      R     DB93.DBX 142.0;
      AN    M 0.7;
      BEC;
      CALL  "STP";
END_ORGANIZATION_BLOCK

ORGANIZATION_BLOCK OB 100
VERSION : 2.3
BEGIN
// (block stored without names or comments; labels and parameter names are numbered)
NETWORK
TITLE =
NETWORK
TITLE =
      SET;
      S     M 0.7;
      R     DB82.DBX 9.6;
      L     0;
      T     DB19.DBB 10;
      CALL  FB 1 , DB 7 (
           DIW 0                    := 1,
           DIW 2                    := 0,
           DID 4                    := P#I 0.0,
           DIW 8                    := 0,
           DID 10                   := P#Q 0.0,
           DIW 14                   := 0,
           DID 16                   := P#Q 8.0,
           DIW 20                   := 0,
           DID 22                   := P#Q 12.0,
           DIW 26                   := 6,
           DIW 28                   := 112,
           DIW 30                   := 32,
           DIW 110                  := 32,
           DIW 112                  := 5376,
           DIX 116.0                := TRUE,
           DIW 118                  := 20,
           DIX 120.0                := TRUE);
NETWORK
TITLE =
      OPN   DB 2;
      L     DBLG;
      T     LW 20;
      L     P#0.0;
      LAR1;
      L     LW 20;
M001: T     LW 20;
      L     0;
      T     DBB [AR1,P#0.0];
      +AR1  P#1.0;
      L     LW 20;
      LOOP  M001;
      OPN   DB 3;
      L     DBLG;
      T     LW 20;
      L     P#0.0;
      LAR1;
      L     LW 20;
M002: T     LW 20;
      L     0;
      T     DBB [AR1,P#0.0];
      +AR1  P#1.0;
      L     LW 20;
      LOOP  M002;
      OPN   DB 92;
      L     DBLG;
      L     40;
      -I;
      T     LW 20;
      L     P#40.0;
      LAR1;
      L     LW 20;
M003: T     LW 20;
      L     0;
      T     DBB [AR1,P#0.0];
      +AR1  P#1.0;
      L     LW 20;
      LOOP  M003;
      OPN   DB 93;
      L     DBLG;
      T     LW 20;
      L     P#0.0;
      LAR1;
      L     LW 20;
M004: T     LW 20;
      L     0;
      T     DBB [AR1,P#0.0];
      +AR1  P#1.0;
      L     LW 20;
      LOOP  M004;
NETWORK
TITLE =
      OPN   DB 97;
      L     DBLG;
      T     LW 20;
      L     P#0.0;
      LAR1;
      L     LW 20;
M005: T     LW 20;
      L     0;
      T     DBB [AR1,P#0.0];
      +AR1  P#1.0;
      L     LW 20;
      LOOP  M005;
      OPN   DB 97;
      L     100;
      T     LW 20;
      L     P#1410.0;
      LAR1;
      L     LW 20;
M006: T     LW 20;
      L     B#16#FF;
      T     DBB [AR1,P#0.0];
      T     DBB [AR1,P#100.0];
      T     DBB [AR1,P#200.0];
      T     DBB [AR1,P#300.0];
      T     DBB [AR1,P#400.0];
      T     DBB [AR1,P#500.0];
      T     DBB [AR1,P#600.0];
      T     DBB [AR1,P#700.0];
      +AR1  P#1.0;
      L     LW 20;
      LOOP  M006;
NETWORK
TITLE =
      L     DB20.DBW 2;
      T     DB90.DBW 0;
      L     DB20.DBW 0;
      T     DB90.DBB 2;
      L     DB20.DBW 20;
      T     DB90.DBW 564;
      SET;
      R     DB90.DBX 172.1;
      R     M 0.7;
END_ORGANIZATION_BLOCK

ORGANIZATION_BLOCK OB 121
VERSION : 0.0
BEGIN
// (block stored without names or comments; labels and parameter names are numbered)
NETWORK
TITLE =
      L     LD 0;
      T     DB93.DBD 0;
      T     DB93.DBD 166;
      L     LD 4;
      T     DB93.DBD 4;
      T     DB93.DBD 170;
      L     LD 8;
      T     DB93.DBD 8;
      T     DB93.DBD 174;
      L     LD 12;
      T     DB93.DBD 12;
      T     DB93.DBD 178;
      L     LD 16;
      T     DB93.DBD 16;
      T     DB93.DBD 182;
      L     121;
      T     DB93.DBD 50;
      SET;
      S     DB93.DBX 164.0;
      AN    M 0.7;
      BEC;
      CALL  "STP";
END_ORGANIZATION_BLOCK

ORGANIZATION_BLOCK OB 122
VERSION : 0.0
BEGIN
// (block stored without names or comments; labels and parameter names are numbered)
NETWORK
TITLE =
      L     LD 0;
      T     DB93.DBD 0;
      T     DB93.DBD 188;
      L     LD 4;
      T     DB93.DBD 4;
      T     DB93.DBD 192;
      L     LD 8;
      T     DB93.DBD 8;
      T     DB93.DBD 196;
      L     LD 12;
      T     DB93.DBD 12;
      T     DB93.DBD 200;
      L     LD 16;
      T     DB93.DBD 16;
      T     DB93.DBD 204;
      L     122;
      T     DB93.DBD 50;
      SET;
      S     DB93.DBX 186.0;
      AN    M 0.7;
      BEC;
      CALL  "STP";
END_ORGANIZATION_BLOCK
